// TwinCAT 3 PLC project TckitUtilsTests
// ProgramVersion: 3.1.4026.22
// libraries:
//   Tc2_Standard, * (Beckhoff Automation GmbH)
//   Tc2_System, * (Beckhoff Automation GmbH)
//   TcUnit, * (www.tcunit.org)
//   T3TckitUtils_Plc,newest,Tc3 Project
// project tree:
//   DUTs/RingBuffer/ ST_Sample.TcDUT
//   / PlcTask.TcTTO
//   POUs/ MAIN.TcPOU
//   POUs/PID/ FB_PidTests.TcPOU
//   POUs/RingBuffer/ FB_RingBufferTests.TcPOU
//   POUs/Strings/ FB_StringTests.TcPOU
// real-time tasks:
//   TASK PlcTask: cycle T#10ms, priority 20, ADS port 350

CONFIGURATION TckitUtilsTests
    RESOURCE PLC ON TwinCAT3
        TASK PlcTask(INTERVAL := T#10ms, PRIORITY := 20);
        PROGRAM MAIN WITH PlcTask : MAIN;
    END_RESOURCE
END_CONFIGURATION

// ---- DUTs/RingBuffer/ST_Sample.TcDUT
TYPE ST_Sample :
STRUCT
    t : LREAL;
    v : LREAL;
END_STRUCT
END_TYPE

// ---- POUs/MAIN.TcPOU
PROGRAM MAIN
VAR
    pidSuite : FB_PidTests;
    rbSuite  : FB_RingBufferTests;
    strSuite : FB_StringTests;
END_VAR

pidSuite();
rbSuite();
strSuite();
TcUnit.RUN();

END_PROGRAM

// ---- POUs/PID/FB_PidTests.TcPOU
FUNCTION_BLOCK FB_PidTests EXTENDS TcUnit.FB_TestSuite
VAR
    pid       : T3TckitUtils_Plc.FB_Pid;
    iPid      : T3TckitUtils_Plc.I_Pid;
    output    : LREAL;
    output2   : LREAL;
    integral  : LREAL;
    saturated : BOOL;
    i         : DINT;
END_VAR

PProportionalOnly();
OutputClampsToMax();
OutputClampsToMin();
IntegralAccumulates();
AntiWindupHoldsIntegral();
DerivativeOnMeasurementNoSetpointSpike();
ReverseModeFlipsSign();
ResetClearsIntegral();
SetterRejectsNegativeKp();
IsSaturatedReflectsClampState();
CyclicReachableThroughInterface();

METHOD AntiWindupHoldsIntegral : BOOL
VAR
    integral : LREAL;
    i : DINT;
END_VAR
IF TEST_ORDERED(__POUNAME()) THEN
    pid.Reset();
    pid.Kp := 0.0;
    pid.Ki := 10.0;
    pid.Kd := 0.0;
    pid.Mode := 0;
    pid.OutputMin := -1.0;
    pid.OutputMax := 1.0;
    FOR i := 1 TO 20 DO
        pid.Update(setpoint := 1.0, measurement := 0.0, deltaT := 0.1);
    END_FOR
    integral := pid.IntegralTerm;
    AssertTrue(Condition := integral <= 0.2,
        Message := 'Anti-windup should hold integral at/near saturation point, not let it grow');
    TEST_FINISHED();
END_IF
END_METHOD

METHOD CyclicReachableThroughInterface : BOOL
VAR
    direct    : LREAL;
    viaIface  : LREAL;
END_VAR
IF TEST_ORDERED(__POUNAME()) THEN
    pid.Reset();
    pid.Kp := 3.0;
    pid.Ki := 0.0;
    pid.Kd := 0.0;
    pid.Mode := 0;
    pid.OutputMin := -100.0;
    pid.OutputMax := 100.0;
    direct := pid.Update(setpoint := 1.0, measurement := 0.0, deltaT := 0.1);

    pid.Reset();
    iPid := pid;
    viaIface := iPid.Update(setpoint := 1.0, measurement := 0.0, deltaT := 0.1);

    AssertEquals_LREAL(Expected := direct, Actual := viaIface, Delta := 1E-9,
        Message := 'Same Update inputs through pid and iPid must give the same output');
    TEST_FINISHED();
END_IF
END_METHOD

METHOD DerivativeOnMeasurementNoSetpointSpike : BOOL
VAR
    output : LREAL;
    output2 : LREAL;
END_VAR
IF TEST_ORDERED(__POUNAME()) THEN
    pid.Reset();
    pid.Kp := 0.0;
    pid.Ki := 0.0;
    pid.Kd := 1.0;
    pid.Mode := 0;
    pid.OutputMin := -100.0;
    pid.OutputMax := 100.0;
    pid.Update(setpoint := 0.0, measurement := 0.0, deltaT := 0.1);
    output := pid.Update(setpoint := 10.0, measurement := 0.0, deltaT := 0.1);
    AssertTrue(Condition := ABS(output) < 1.0,
        Message := 'Derivative-on-measurement: setpoint step must NOT cause D-kick');
    TEST_FINISHED();
END_IF
END_METHOD

METHOD IntegralAccumulates : BOOL
VAR
    integral : LREAL;
    i : DINT;
END_VAR
IF TEST_ORDERED(__POUNAME()) THEN
    pid.Reset();
    pid.Kp := 0.0;
    pid.Ki := 1.0;
    pid.Kd := 0.0;
    pid.Mode := 0;
    pid.OutputMin := -100.0;
    pid.OutputMax := 100.0;
    FOR i := 1 TO 10 DO
        pid.Update(setpoint := 1.0, measurement := 0.0, deltaT := 0.1);
    END_FOR
    integral := pid.IntegralTerm;
    AssertEquals_LREAL(Expected := 1.0, Actual := integral, Delta := 0.05,
        Message := 'I-only Ki=1 error=1 for 10x0.1s should integrate to ~1.0');
    TEST_FINISHED();
END_IF
END_METHOD

METHOD IsSaturatedReflectsClampState : BOOL
VAR
    saturated : BOOL;
END_VAR
IF TEST_ORDERED(__POUNAME()) THEN
    pid.Reset();
    pid.Kp := 1.0;
    pid.Ki := 0.0;
    pid.Kd := 0.0;
    pid.Mode := 0;
    pid.OutputMin := -10.0;
    pid.OutputMax := 10.0;
    pid.Update(setpoint := 1.0, measurement := 0.0, deltaT := 0.1);
    saturated := pid.IsSaturated;
    AssertFalse(Condition := saturated,
        Message := 'IsSaturated should be FALSE when output is within OutputMin..OutputMax');
    pid.Update(setpoint := 100.0, measurement := 0.0, deltaT := 0.1);
    saturated := pid.IsSaturated;
    AssertTrue(Condition := saturated,
        Message := 'IsSaturated should be TRUE once the output is clamped to OutputMax');
    TEST_FINISHED();
END_IF
END_METHOD

METHOD OutputClampsToMax : BOOL
VAR
    output : LREAL;
END_VAR
IF TEST_ORDERED(__POUNAME()) THEN
    pid.Reset();
    pid.Kp := 2.0;
    pid.Ki := 0.0;
    pid.Kd := 0.0;
    pid.Mode := 0;
    pid.OutputMin := -5.0;
    pid.OutputMax := 5.0;
    output := pid.Update(setpoint := 100.0, measurement := 0.0, deltaT := 0.1);
    AssertEquals_LREAL(Expected := 5.0, Actual := output, Delta := 1E-6,
        Message := 'Output should clamp to OutputMax on large positive error');
    TEST_FINISHED();
END_IF
END_METHOD

METHOD OutputClampsToMin : BOOL
VAR
    output : LREAL;
END_VAR
IF TEST_ORDERED(__POUNAME()) THEN
    pid.Reset();
    pid.Kp := 2.0;
    pid.Ki := 0.0;
    pid.Kd := 0.0;
    pid.Mode := 0;
    pid.OutputMin := -5.0;
    pid.OutputMax := 5.0;
    output := pid.Update(setpoint := -100.0, measurement := 0.0, deltaT := 0.1);
    AssertEquals_LREAL(Expected := -5.0, Actual := output, Delta := 1E-6,
        Message := 'Output should clamp to OutputMin on large negative error');
    TEST_FINISHED();
END_IF
END_METHOD

METHOD PProportionalOnly : BOOL
VAR
    output : LREAL;
END_VAR
IF TEST_ORDERED(__POUNAME()) THEN
    pid.Reset();
    pid.Kp := 2.0;
    pid.Ki := 0.0;
    pid.Kd := 0.0;
    pid.Mode := 0;
    pid.OutputMin := -100.0;
    pid.OutputMax := 100.0;
    output := pid.Update(setpoint := 1.0, measurement := 0.0, deltaT := 0.1);
    AssertEquals_LREAL(Expected := 2.0, Actual := output, Delta := 1E-6,
        Message := 'P-only Kp=2 error=1 should yield output=2');
    TEST_FINISHED();
END_IF
END_METHOD

METHOD ResetClearsIntegral : BOOL
VAR
    integral : LREAL;
    i : DINT;
END_VAR
IF TEST_ORDERED(__POUNAME()) THEN
    pid.Kp := 0.0;
    pid.Ki := 1.0;
    pid.Kd := 0.0;
    pid.Mode := 0;
    pid.OutputMin := -100.0;
    pid.OutputMax := 100.0;
    FOR i := 1 TO 5 DO
        pid.Update(setpoint := 1.0, measurement := 0.0, deltaT := 0.1);
    END_FOR
    AssertTrue(Condition := pid.IntegralTerm > 0.0,
        Message := 'Integral must be non-zero before Reset for this test to be meaningful');
    pid.Reset();
    integral := pid.IntegralTerm;
    AssertEquals_LREAL(Expected := 0.0, Actual := integral, Delta := 1E-9,
        Message := 'Reset must zero the integral term');
    TEST_FINISHED();
END_IF
END_METHOD

METHOD ReverseModeFlipsSign : BOOL
VAR
    output : LREAL;
END_VAR
IF TEST_ORDERED(__POUNAME()) THEN
    pid.Reset();
    pid.Kp := 2.0;
    pid.Ki := 0.0;
    pid.Kd := 0.0;
    pid.Mode := 1;
    pid.OutputMin := -100.0;
    pid.OutputMax := 100.0;
    output := pid.Update(setpoint := 1.0, measurement := 0.0, deltaT := 0.1);
    AssertEquals_LREAL(Expected := -2.0, Actual := output, Delta := 1E-6,
        Message := 'Reverse mode should flip the sign of the controller output');
    TEST_FINISHED();
END_IF
END_METHOD

METHOD SetterRejectsNegativeKp : BOOL
IF TEST_ORDERED(__POUNAME()) THEN
    pid.Kp := 0.5;
    pid.Kp := -1.0;
    AssertEquals_LREAL(Expected := 0.5, Actual := pid.Kp, Delta := 1E-9,
        Message := 'Setter must reject negative Kp; existing value preserved');
    TEST_FINISHED();
END_IF
END_METHOD

END_FUNCTION_BLOCK

// ---- POUs/RingBuffer/FB_RingBufferTests.TcPOU
FUNCTION_BLOCK FB_RingBufferTests EXTENDS TcUnit.FB_TestSuite
VAR
END_VAR

ConfigureRejectsZeroCapacity();
EmptyAfterConfigure();
PushPopFifoLreal();
PushPopFifoInt();
PushPopUserDefinedStruct();
PeekDoesNotConsume();
WrapAroundPreservesOrder();
PushReturnsFalseWhenFull();
PopReturnsFalseWhenEmpty();

METHOD ConfigureRejectsZeroCapacity : BOOL
VAR
    rb       : T3TckitUtils_Plc.FB_RingBuffer;
    storage  : ARRAY[1..4] OF LREAL;
END_VAR
IF TEST_ORDERED(__POUNAME()) THEN
    AssertFalse(Condition := rb.Configure(storage, 0),
        Message := 'Configure with capacity=0 must return FALSE');
    AssertTrue(Condition := rb.Configure(storage, 4),
        Message := 'Configure with matched diSize/capacity must return TRUE');
    TEST_FINISHED();
END_IF
END_METHOD

METHOD EmptyAfterConfigure : BOOL
VAR
    rb       : T3TckitUtils_Plc.FB_RingBuffer;
    storage  : ARRAY[1..4] OF LREAL;
END_VAR
IF TEST_ORDERED(__POUNAME()) THEN
    AssertTrue(Condition := rb.Configure(storage, 4),
        Message := 'Configure must succeed for ARRAY[1..4] OF LREAL with capacity=4');
    AssertEquals_UDINT(Expected := 0, Actual := rb.Count,
        Message := 'Fresh buffer Count must be 0');
    AssertTrue(Condition := rb.IsEmpty,
        Message := 'Fresh buffer IsEmpty must be TRUE');
    AssertFalse(Condition := rb.IsFull,
        Message := 'Fresh buffer IsFull must be FALSE');
    AssertEquals_UDINT(Expected := 4, Actual := rb.Capacity,
        Message := 'Capacity must reflect the configured value');
    TEST_FINISHED();
END_IF
END_METHOD

METHOD PeekDoesNotConsume : BOOL
VAR
    rb       : T3TckitUtils_Plc.FB_RingBuffer;
    storage  : ARRAY[1..4] OF LREAL;
    v1       : LREAL;
    seen     : LREAL;
END_VAR
IF TEST_ORDERED(__POUNAME()) THEN
    rb.Configure(storage, 4);
    v1 := 7.5;
    rb.Push(v1);
    AssertTrue(Condition := rb.Peek(seen),
        Message := 'Peek must succeed when buffer is non-empty');
    AssertEquals_LREAL(Expected := 7.5, Actual := seen, Delta := 1E-9,
        Message := 'Peek must return the front element');
    AssertEquals_UDINT(Expected := 1, Actual := rb.Count,
        Message := 'Peek must not change Count');
    seen := 0.0;
    rb.Peek(seen);
    AssertEquals_LREAL(Expected := 7.5, Actual := seen, Delta := 1E-9,
        Message := 'A second Peek must return the same element');
    TEST_FINISHED();
END_IF
END_METHOD

METHOD PopReturnsFalseWhenEmpty : BOOL
VAR
    rb       : T3TckitUtils_Plc.FB_RingBuffer;
    storage  : ARRAY[1..4] OF LREAL;
    popped   : LREAL;
END_VAR
IF TEST_ORDERED(__POUNAME()) THEN
    rb.Configure(storage, 4);
    AssertFalse(Condition := rb.Pop(popped),
        Message := 'Pop must return FALSE on an empty buffer');
    AssertFalse(Condition := rb.Peek(popped),
        Message := 'Peek must return FALSE on an empty buffer');
    TEST_FINISHED();
END_IF
END_METHOD

METHOD PushPopFifoInt : BOOL
VAR
    rb       : T3TckitUtils_Plc.FB_RingBuffer;
    storage  : ARRAY[1..4] OF INT;
    v1, v2   : INT;
    popped   : INT;
END_VAR
IF TEST_ORDERED(__POUNAME()) THEN
    rb.Configure(storage, 4);
    v1 := 11;
    v2 := 22;
    rb.Push(v1);
    rb.Push(v2);
    AssertEquals_UDINT(Expected := 2, Actual := rb.Count,
        Message := 'Count after two INT pushes must be 2');
    rb.Pop(popped);
    AssertEquals_INT(Expected := 11, Actual := popped,
        Message := 'INT FIFO order must match LREAL FIFO order');
    rb.Pop(popped);
    AssertEquals_INT(Expected := 22, Actual := popped,
        Message := 'Second INT Pop must return the second Push');
    TEST_FINISHED();
END_IF
END_METHOD

METHOD PushPopFifoLreal : BOOL
VAR
    rb       : T3TckitUtils_Plc.FB_RingBuffer;
    storage  : ARRAY[1..4] OF LREAL;
    v1, v2, v3 : LREAL;
    popped   : LREAL;
END_VAR
IF TEST_ORDERED(__POUNAME()) THEN
    rb.Configure(storage, 4);
    v1 := 1.0;
    v2 := 2.0;
    v3 := 3.0;
    AssertTrue(Condition := rb.Push(v1), Message := 'Push(1.0) must succeed');
    AssertTrue(Condition := rb.Push(v2), Message := 'Push(2.0) must succeed');
    AssertTrue(Condition := rb.Push(v3), Message := 'Push(3.0) must succeed');
    AssertEquals_UDINT(Expected := 3, Actual := rb.Count,
        Message := 'Count after three pushes must be 3');
    AssertTrue(Condition := rb.Pop(popped), Message := 'Pop must succeed when buffer is non-empty');
    AssertEquals_LREAL(Expected := 1.0, Actual := popped, Delta := 1E-9,
        Message := 'First Pop must return the first Push');
    rb.Pop(popped);
    AssertEquals_LREAL(Expected := 2.0, Actual := popped, Delta := 1E-9,
        Message := 'Second Pop must return the second Push');
    rb.Pop(popped);
    AssertEquals_LREAL(Expected := 3.0, Actual := popped, Delta := 1E-9,
        Message := 'Third Pop must return the third Push');
    AssertTrue(Condition := rb.IsEmpty,
        Message := 'Buffer must be empty after popping all elements');
    TEST_FINISHED();
END_IF
END_METHOD

METHOD PushPopUserDefinedStruct : BOOL
VAR
    rb       : T3TckitUtils_Plc.FB_RingBuffer;
    storage  : ARRAY[1..4] OF ST_Sample;
    inA, inB : ST_Sample;
    popped   : ST_Sample;
END_VAR
IF TEST_ORDERED(__POUNAME()) THEN
    rb.Configure(storage, 4);
    inA.t := 0.1; inA.v := 11.0;
    inB.t := 0.2; inB.v := 22.0;
    rb.Push(inA);
    rb.Push(inB);
    AssertEquals_UDINT(Expected := 2, Actual := rb.Count,
        Message := 'Count after two ST_Sample pushes must be 2');
    rb.Pop(popped);
    AssertEquals_LREAL(Expected := 0.1, Actual := popped.t, Delta := 1E-9,
        Message := 'ST_Sample.t must round-trip exactly');
    AssertEquals_LREAL(Expected := 11.0, Actual := popped.v, Delta := 1E-9,
        Message := 'ST_Sample.v must round-trip exactly');
    rb.Pop(popped);
    AssertEquals_LREAL(Expected := 0.2, Actual := popped.t, Delta := 1E-9,
        Message := 'Second ST_Sample.t must round-trip exactly');
    AssertEquals_LREAL(Expected := 22.0, Actual := popped.v, Delta := 1E-9,
        Message := 'Second ST_Sample.v must round-trip exactly');
    TEST_FINISHED();
END_IF
END_METHOD

METHOD PushReturnsFalseWhenFull : BOOL
VAR
    rb       : T3TckitUtils_Plc.FB_RingBuffer;
    storage  : ARRAY[1..2] OF LREAL;
    v1, v2, v3 : LREAL;
END_VAR
IF TEST_ORDERED(__POUNAME()) THEN
    rb.Configure(storage, 2);
    v1 := 1.0; v2 := 2.0; v3 := 3.0;
    AssertTrue(Condition := rb.Push(v1), Message := 'First Push must succeed');
    AssertTrue(Condition := rb.Push(v2), Message := 'Second Push must succeed');
    AssertTrue(Condition := rb.IsFull,
        Message := 'IsFull must be TRUE when Count = Capacity');
    AssertFalse(Condition := rb.Push(v3),
        Message := 'Push must return FALSE when the buffer is full');
    AssertEquals_UDINT(Expected := 2, Actual := rb.Count,
        Message := 'A refused Push must not change Count');
    TEST_FINISHED();
END_IF
END_METHOD

METHOD WrapAroundPreservesOrder : BOOL
VAR
    rb       : T3TckitUtils_Plc.FB_RingBuffer;
    storage  : ARRAY[1..3] OF LREAL;
    a, b, c, d, e : LREAL;
    popped   : LREAL;
END_VAR
IF TEST_ORDERED(__POUNAME()) THEN
    rb.Configure(storage, 3);
    a := 1.0; b := 2.0; c := 3.0;
    rb.Push(a); rb.Push(b); rb.Push(c);
    rb.Pop(popped);
    AssertEquals_LREAL(Expected := 1.0, Actual := popped, Delta := 1E-9,
        Message := 'First Pop must return 1.0 before wrap');
    rb.Pop(popped);
    AssertEquals_LREAL(Expected := 2.0, Actual := popped, Delta := 1E-9,
        Message := 'Second Pop must return 2.0 before wrap');
    d := 4.0; e := 5.0;
    AssertTrue(Condition := rb.Push(d),
        Message := 'Push after Pops must succeed (forces write index to wrap)');
    AssertTrue(Condition := rb.Push(e),
        Message := 'Second Push after Pops must also succeed');
    rb.Pop(popped);
    AssertEquals_LREAL(Expected := 3.0, Actual := popped, Delta := 1E-9,
        Message := 'After wrap, Pop must return 3.0 (the surviving pre-wrap element)');
    rb.Pop(popped);
    AssertEquals_LREAL(Expected := 4.0, Actual := popped, Delta := 1E-9,
        Message := 'After wrap, second Pop must return 4.0');
    rb.Pop(popped);
    AssertEquals_LREAL(Expected := 5.0, Actual := popped, Delta := 1E-9,
        Message := 'After wrap, third Pop must return 5.0');
    TEST_FINISHED();
END_IF
END_METHOD

END_FUNCTION_BLOCK

// ---- POUs/Strings/FB_StringTests.TcPOU
FUNCTION_BLOCK FB_StringTests EXTENDS TcUnit.FB_TestSuite
VAR
END_VAR

BuilderEmptyOnInit();
BuilderAppendOnce();
BuilderAppendMany();
BuilderAppendOverflowReturnsFalse();
BuilderClearResetsLength();
TrimStripsSurroundingWhitespace();
StartsWithEndsWithBoundaries();
ContainsFindsSubstring();

METHOD BuilderAppendMany : BOOL
VAR
    sb : T3TckitUtils_Plc.FB_StringBuilder;
    i  : DINT;
    ok : BOOL;
END_VAR
IF TEST_ORDERED(__POUNAME()) THEN
    ok := TRUE;
    FOR i := 1 TO 500 DO
        ok := ok AND sb.Append('ab');
    END_FOR
    AssertTrue(Condition := ok,
        Message := 'Each of the 500 two-byte appends must succeed (1000 < 4095)');
    AssertEquals_UDINT(Expected := 1000, Actual := sb.Length,
        Message := 'Length after 500 x "ab" must be 1000');
    AssertFalse(Condition := sb.IsFull,
        Message := 'IsFull must remain FALSE while Length < Capacity');
    TEST_FINISHED();
END_IF
END_METHOD

METHOD BuilderAppendOnce : BOOL
VAR
    sb       : T3TckitUtils_Plc.FB_StringBuilder;
    buf      : ARRAY[1..32] OF BYTE;
    written  : UDINT;
END_VAR
IF TEST_ORDERED(__POUNAME()) THEN
    AssertTrue(Condition := sb.Append('hello'),
        Message := 'Append("hello") must succeed on an empty builder');
    AssertEquals_UDINT(Expected := 5, Actual := sb.Length,
        Message := 'Length after Append("hello") must be 5');
    written := sb.CopyTo(ADR(buf), SIZEOF(buf));
    AssertEquals_UDINT(Expected := 5, Actual := written,
        Message := 'CopyTo must report 5 payload bytes');
    AssertEquals_BYTE(Expected := 16#68, Actual := buf[1],
        Message := 'First copied byte must be ASCII "h" (0x68)');
    AssertEquals_BYTE(Expected := 16#6F, Actual := buf[5],
        Message := 'Fifth copied byte must be ASCII "o" (0x6F)');
    TEST_FINISHED();
END_IF
END_METHOD

METHOD BuilderAppendOverflowReturnsFalse : BOOL
VAR
    sb        : T3TckitUtils_Plc.FB_StringBuilder;
    i         : DINT;
    rejected  : BOOL;
    lengthAt  : UDINT;
END_VAR
IF TEST_ORDERED(__POUNAME()) THEN
    rejected := FALSE;
    FOR i := 1 TO 4100 DO
        IF NOT sb.Append('X') THEN
            rejected := TRUE;
            lengthAt := sb.Length;
            EXIT;
        END_IF
    END_FOR
    AssertTrue(Condition := rejected,
        Message := 'A single-byte Append must return FALSE before 4100 calls have completed');
    AssertEquals_UDINT(Expected := 4095, Actual := lengthAt,
        Message := 'Length at refusal point must equal Capacity (4095)');
    AssertTrue(Condition := sb.IsFull,
        Message := 'IsFull must be TRUE at the refusal point');
    TEST_FINISHED();
END_IF
END_METHOD

METHOD BuilderClearResetsLength : BOOL
VAR
    sb : T3TckitUtils_Plc.FB_StringBuilder;
END_VAR
IF TEST_ORDERED(__POUNAME()) THEN
    sb.Append('payload');
    AssertTrue(Condition := sb.Length > 0,
        Message := 'Builder must have non-zero Length before Clear for the test to be meaningful');
    sb.Clear();
    AssertEquals_UDINT(Expected := 0, Actual := sb.Length,
        Message := 'Clear must zero Length');
    AssertTrue(Condition := sb.Append('again'),
        Message := 'Append after Clear must succeed');
    AssertEquals_UDINT(Expected := 5, Actual := sb.Length,
        Message := 'Length must reflect the post-Clear Append');
    TEST_FINISHED();
END_IF
END_METHOD

METHOD BuilderEmptyOnInit : BOOL
VAR
    sb : T3TckitUtils_Plc.FB_StringBuilder;
END_VAR
IF TEST_ORDERED(__POUNAME()) THEN
    AssertEquals_UDINT(Expected := 0, Actual := sb.Length,
        Message := 'Freshly constructed builder Length must be 0');
    AssertFalse(Condition := sb.IsFull,
        Message := 'Freshly constructed builder IsFull must be FALSE');
    AssertEquals_UDINT(Expected := 4095, Actual := sb.Capacity,
        Message := 'Builder Capacity must be the documented 4095 bytes');
    TEST_FINISHED();
END_IF
END_METHOD

METHOD ContainsFindsSubstring : BOOL
IF TEST_ORDERED(__POUNAME()) THEN
    AssertTrue(Condition := T3TckitUtils_Plc.F_Contains('one two three', 'two'),
        Message := 'F_Contains must find an interior substring');
    AssertFalse(Condition := T3TckitUtils_Plc.F_Contains('abc', 'd'),
        Message := 'F_Contains must return FALSE when the needle is absent');
    AssertTrue(Condition := T3TckitUtils_Plc.F_Contains('any', ''),
        Message := 'F_Contains with an empty needle must return TRUE');
    AssertFalse(Condition := T3TckitUtils_Plc.F_Contains('', 'x'),
        Message := 'F_Contains over an empty string must return FALSE for a non-empty needle');
    TEST_FINISHED();
END_IF
END_METHOD

METHOD StartsWithEndsWithBoundaries : BOOL
IF TEST_ORDERED(__POUNAME()) THEN
    AssertTrue(Condition := T3TckitUtils_Plc.F_StartsWith('foobar', 'foo'),
        Message := 'F_StartsWith must return TRUE for a matching prefix');
    AssertFalse(Condition := T3TckitUtils_Plc.F_StartsWith('foo', 'foobar'),
        Message := 'F_StartsWith must return FALSE when the prefix is longer than the string');
    AssertTrue(Condition := T3TckitUtils_Plc.F_StartsWith('anything', ''),
        Message := 'F_StartsWith with an empty prefix must return TRUE');
    AssertTrue(Condition := T3TckitUtils_Plc.F_EndsWith('foobar', 'bar'),
        Message := 'F_EndsWith must return TRUE for a matching suffix');
    AssertFalse(Condition := T3TckitUtils_Plc.F_EndsWith('bar', 'foobar'),
        Message := 'F_EndsWith must return FALSE when the suffix is longer than the string');
    AssertTrue(Condition := T3TckitUtils_Plc.F_EndsWith('anything', ''),
        Message := 'F_EndsWith with an empty suffix must return TRUE');
    TEST_FINISHED();
END_IF
END_METHOD

METHOD TrimStripsSurroundingWhitespace : BOOL
IF TEST_ORDERED(__POUNAME()) THEN
    AssertEquals_STRING(Expected := 'hi', Actual := T3TckitUtils_Plc.F_Trim('  hi  '),
        Message := 'F_Trim must strip surrounding spaces');
    AssertEquals_STRING(Expected := 'hi', Actual := T3TckitUtils_Plc.F_Trim('$Thi$N'),
        Message := 'F_Trim must strip tab/CR/LF as well as space');
    AssertEquals_STRING(Expected := '', Actual := T3TckitUtils_Plc.F_Trim(''),
        Message := 'F_Trim of the empty string must return the empty string');
    AssertEquals_STRING(Expected := 'inner space', Actual := T3TckitUtils_Plc.F_Trim('inner space'),
        Message := 'F_Trim must preserve internal whitespace');
    TEST_FINISHED();
END_IF
END_METHOD

END_FUNCTION_BLOCK
